// TIA Portal V18 export
FUNCTION "MR_Quantity Control" : Void   // FC16, LAD
{ S7_Optimized_Access := 'TRUE' }
VERSION : 0.1
// stored: AutoNumber true, IsIECCheckEnabled false, SetENOAutomatically false, UDAEnableTagReadback false
   VAR_TEMP
      temp : Bool;
   END_VAR
BEGIN

REGION Network 1 (SCL)
       //IF "Function Ratio check".input.Mode = 0 THEN
           "Function Ratio check".PumpCaliberationControls.CurrentSet_A := (100 / ("Mixing ratio"."Mixing ratio according to density" + real#100)) * "Function Ratio check".input."set qty";
         "Function Ratio check".PumpCaliberationControls.CurrentSet_B := "Function Ratio check".input."set qty" - "Function Ratio check".PumpCaliberationControls.CurrentSet_A;
      // END_IF;

       // IF "Function Ratio check".input.Mode = 1 THEN
       //     "Function Ratio check".PumpCaliberationControls.CurrentSet_A := "Function Ratio check".input."set qty";
       //    // "Function Ratio check".PumpCaliberationControls.CurrentSet_B := 0;
       //   //"Function Ratio check".PumpCaliberationControls.CurrentSet_B := "Function Ratio check".input."set qty" - "Function Ratio check".PumpCaliberationControls.CurrentSet_A;
       // END_IF;

       // IF "Function Ratio check".input.Mode = 2 THEN
       //  // "Function Ratio check".PumpCaliberationControls.CurrentSet_A := 0;
       //   "Function Ratio check".PumpCaliberationControls.CurrentSet_B := "Function Ratio check".input."set qty";//- "Function Ratio check".PumpCaliberationControls.CurrentSet_A;
       // END_IF;


       //Progress bar Higher limit for Ratio check to display on the screen.
       "Function Ratio check".Control.ProgressBar_Limit := REAL_TO_DINT(("Function Ratio check".input."set qty" / "Function Ratio check".input."Set Flowrate") * 60000);

       // Actual progress bar display on the screen for Ratio check progress.
       "Function Ratio check".Control.ProgressBar := "Function Ratio check".output."Running time" * 1000;
END_REGION

REGION Network 2
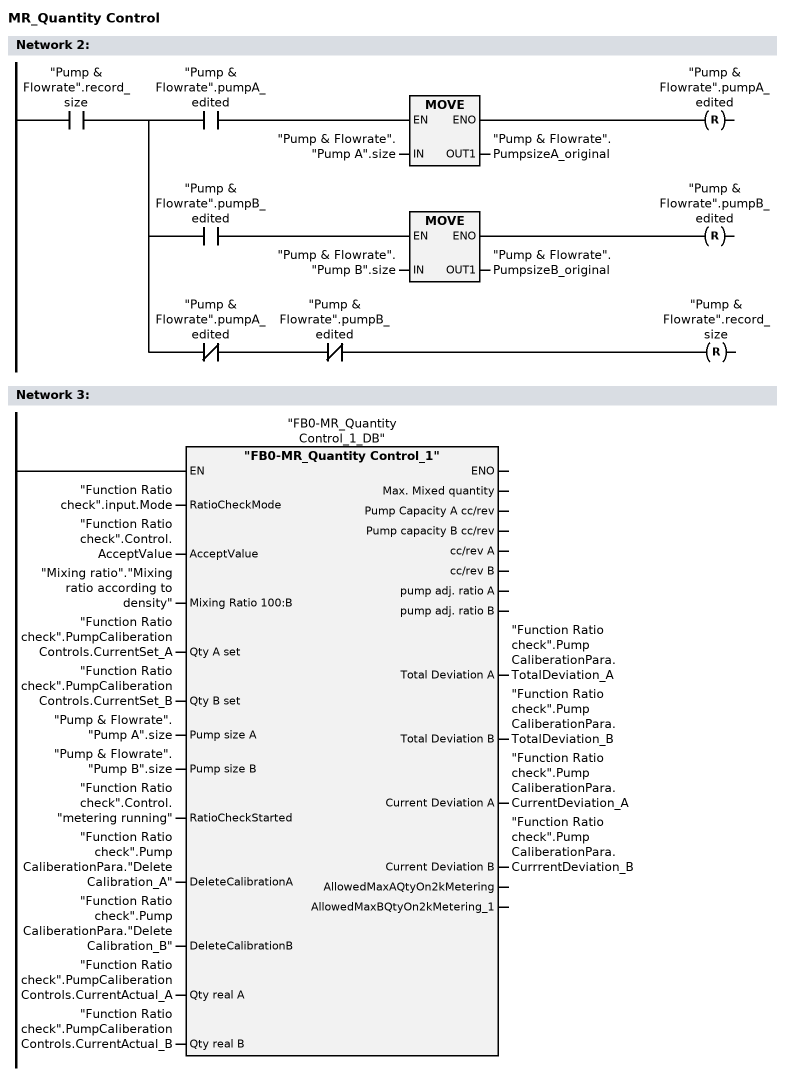
   IF "Pump & Flowrate".record_size AND "Pump & Flowrate".pumpA_edited THEN
       "Pump & Flowrate".PumpsizeA_original := "Pump & Flowrate"."Pump A".size;
       "Pump & Flowrate".pumpA_edited := FALSE;
   END_IF;
   IF "Pump & Flowrate".record_size AND "Pump & Flowrate".pumpB_edited THEN
       "Pump & Flowrate".PumpsizeB_original := "Pump & Flowrate"."Pump B".size;
       "Pump & Flowrate".pumpB_edited := FALSE;
   END_IF;
   IF "Pump & Flowrate".record_size AND NOT "Pump & Flowrate".pumpA_edited AND NOT "Pump & Flowrate".pumpB_edited THEN
       "Pump & Flowrate".record_size := FALSE;
   END_IF;
END_REGION

REGION Network 3
   RUNG wire#powerrail
      "FB0-MR_Quantity Control_1_DB"(RatioCheckMode := "Function Ratio check".input.Mode, AcceptValue := "Function Ratio check".Control.AcceptValue, "Mixing Ratio 100:B" := "Mixing ratio"."Mixing ratio according to density", "Qty A set" := "Function Ratio check".PumpCaliberationControls.CurrentSet_A, "Qty B set" := "Function Ratio check".PumpCaliberationControls.CurrentSet_B, "Pump size A" := "Pump & Flowrate"."Pump A".size, "Pump size B" := "Pump & Flowrate"."Pump B".size, RatioCheckStarted := "Function Ratio check".Control."metering running", DeleteCalibrationA := "Function Ratio check".PumpCaliberationPara."Delete Calibration_A", DeleteCalibrationB := "Function Ratio check".PumpCaliberationPara."Delete Calibration_B", "Qty real A" := "Function Ratio check".PumpCaliberationControls.CurrentActual_A, "Qty real B" := "Function Ratio check".PumpCaliberationControls.CurrentActual_B, "Max. Mixed quantity" =>, "Pump Capacity A cc/rev" =>, "Pump capacity B cc/rev" =>, "cc/rev A" =>, "cc/rev B" =>, "pump adj. ratio A" =>, "pump adj. ratio B" =>, "Total Deviation A" => "Function Ratio check".PumpCaliberationPara.TotalDeviation_A, "Total Deviation B" => "Function Ratio check".PumpCaliberationPara.TotalDeviation_B, "Current Deviation A" => "Function Ratio check".PumpCaliberationPara.CurrentDeviation_A, "Current Deviation B" => "Function Ratio check".PumpCaliberationPara.CurrrentDeviation_B, AllowedMaxAQtyOn2kMetering =>, AllowedMaxBQtyOn2kMetering_1 =>)
   END_RUNG
   // the same network as SCL:
   "FB0-MR_Quantity Control_1_DB"(RatioCheckMode := "Function Ratio check".input.Mode,   // "FB0-MR_Quantity Control_1"
                           AcceptValue := "Function Ratio check".Control.AcceptValue,
                           "Mixing Ratio 100:B" := "Mixing ratio"."Mixing ratio according to density",
                           "Qty A set" := "Function Ratio check".PumpCaliberationControls.CurrentSet_A,
                           "Qty B set" := "Function Ratio check".PumpCaliberationControls.CurrentSet_B,
                           "Pump size A" := "Pump & Flowrate"."Pump A".size,
                           "Pump size B" := "Pump & Flowrate"."Pump B".size,
                           RatioCheckStarted := "Function Ratio check".Control."metering running",
                           DeleteCalibrationA := "Function Ratio check".PumpCaliberationPara."Delete Calibration_A",
                           DeleteCalibrationB := "Function Ratio check".PumpCaliberationPara."Delete Calibration_B",
                           "Qty real A" := "Function Ratio check".PumpCaliberationControls.CurrentActual_A,
                           "Qty real B" := "Function Ratio check".PumpCaliberationControls.CurrentActual_B,
                           "Total Deviation A" => "Function Ratio check".PumpCaliberationPara.TotalDeviation_A,
                           "Total Deviation B" => "Function Ratio check".PumpCaliberationPara.TotalDeviation_B,
                           "Current Deviation A" => "Function Ratio check".PumpCaliberationPara.CurrentDeviation_A,
                           "Current Deviation B" => "Function Ratio check".PumpCaliberationPara.CurrrentDeviation_B);
END_REGION
END_FUNCTION
